# EPICS substitutions: viocs/si_ps/si_psApp/Db/qdp1.substitutions
file "db/individual.db" {
    pattern { family, pos, num }
        { "QDP1", "03M1", "" }
        { "QDP1", "03M2", "" }
        { "QDP1", "07M1", "" }
        { "QDP1", "07M2", "" }
        { "QDP1", "11M1", "" }
        { "QDP1", "11M2", "" }
        { "QDP1", "15M1", "" }
        { "QDP1", "15M2", "" }
        { "QDP1", "19M1", "" }
        { "QDP1", "19M2", "" }
}
